//{attribute 'qualified_only'}
//{attribute 'strict'}
TYPE E_Door :
(
	eDoor_none := 0,
	
	eDoor_nMaxIdx	
);
END_TYPE

(* stored: Version 1.1.0.1, ProductVersion 3.1.4024.12
   DUT E_Door: Id {bbb1acd8-2e3d-4471-ad73-4e04c672e7a3} *)
